PROGRAM PRG_LoadcellScaling
VAR
END_VAR

GVL.uLoadCellScaledValue := F_Scale(GVL.uLoadCellRawValue, 0.0, 1.0, -383, 1200);

END_PROGRAM

(* stored: Version 1.1.0.1, ProductVersion 3.1.4024.12
   POU PRG_LoadcellScaling: Id {976f5398-c837-4944-8db6-b5f1f3ab8dcc}, SpecialFunc None *)
